// TIA Portal V18 export
TYPE "ST_Stopper"
// stored: IsFailsafeCompliant false
   STRUCT
      ReleasePB : Bool;   // 手动释放按钮
      NoClear : Bool;   // 手动中
      Sensor : Bool;   // 托盘到位
      AutoTrg : Bool;   // 释放
      Done : Bool;   // 完成
      ReleaseFault : Bool;   // 释放异常
      ReachFault : Bool;   // 下站接受异常
   END_STRUCT;
END_TYPE
